SUBAPPLICATION QX_Emulated_SA (* Subapplication Type *)
  (* Standard: 61499-2 *)
  (* Version 1.0, 2023-10-26, kirill *)
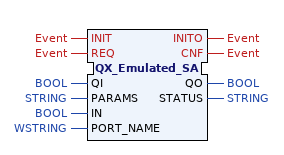
  EVENT_INPUT
    INIT;
    REQ;
  END_EVENT
  EVENT_OUTPUT
    INITO;
    CNF;
  END_EVENT
  VAR_INPUT
    QI : BOOL;
    PARAMS : STRING;
    IN : BOOL;
    PORT_NAME : WSTRING;
  END_VAR
  VAR_OUTPUT
    QO : BOOL;
    STATUS : STRING;
  END_VAR
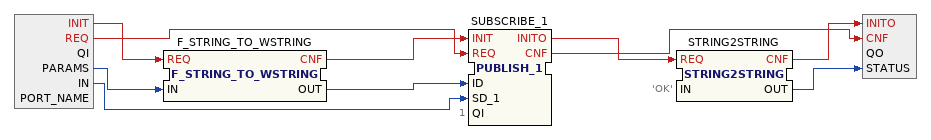
  FBS
    STRING2STRING : STRING2STRING(IN := 'OK');
    SUBSCRIBE_1 : PUBLISH_1(QI := 1);
    F_STRING_TO_WSTRING : F_STRING_TO_WSTRING;
  END_FBS
  EVENT_CONNECTIONS
    SUBSCRIBE_1.INITO TO STRING2STRING.REQ;
    F_STRING_TO_WSTRING.CNF TO SUBSCRIBE_1.INIT;
    INIT TO F_STRING_TO_WSTRING.REQ;
    STRING2STRING.CNF TO INITO;
    SUBSCRIBE_1.CNF TO CNF;
    REQ TO SUBSCRIBE_1.REQ;
  END_CONNECTIONS
  DATA_CONNECTIONS
    F_STRING_TO_WSTRING.OUT TO SUBSCRIBE_1.ID;
    PARAMS TO F_STRING_TO_WSTRING.IN;
    STRING2STRING.OUT TO STATUS;
    IN TO SUBSCRIBE_1.SD_1;
  END_CONNECTIONS
END_SUBAPPLICATION
